(* Logix 5000 project; controller Transcat_L33ER vendor 1 type 14 code 107 rev 32.11; software revision 32.02; part 3 of 5 *)
(* tags used below, declared in another part *)
   AcsiiToReal1 : HexASCII_to_REAL;
   ActiveRecipe : Recipe;   // Active process recipe downloaded from the HMI recipe system and used by the PLC for automatic operation.
   AllDevice1stScanDone : BOOL;   // When this bit is set - all devices have been scanned once and bits reset
   AllDeviceEnable : BOOL;   // A bit to enable or disable the running of all devices
   AllReset : BOOL;   // Bit to reset Auto/Man, AutoRun, RecipeRun, TimedRunEnable to 0 from PLC
   alwaysOFF : BOOL;
   AnyAutoRun : BOOL;   // Bit that in on if ANY device is placed into Auto run (to signal pre-start beed)
   AnyAutoRunFlag : BOOL;   // A flag that indicates if any device is in Auto Run (used with pre-start beep logic)
   AnyManRunFlag : BOOL;   // A flag that indicates if any device is in Manual Run (used with pre-start beep logic)
   AnyManualRun : BOOL;   // Bit that in on if ANY device is placed into manual run (to signal pre-start beed)
   Auto_Run_All_Interlock : BOOL;   // Bit to interlock all devices running in Auto
   AutoRunRequest : BOOL;   // True when the automatic state machine is in RUNNING and automatic device operation is requested.
   Beep : BOOL;   // Bit to Activte Beacon Alarm
   bronkhorstReal : REAL[50];   // data from Bonkhorst - convertred to real values
   BronkOutArr : DINT[3];   // 3 Outputs from Flow controllers 0 - 100% = 0 - 32000
   BronkRealInArr : REAL[100];
   ConversionError : BOOL;
   ConvertedFloat : REAL;
   dataIndex : DINT;   // Bronkhorst Data Index
   Device : Device[20];
   DiscreteTemp : BOOL;   // A temporay boolean to hold positions during PLC transer
   dNum : DINT;   // The index of the current device being processed
   DoseCounter : COUNTER;   // Counts the # of doses since last reset
   DoseCounterReset_HMI : BOOL;   // HMI bit to reset the dose counter
   DoseStart : BOOL;   // Bit to start dosing sequence
   DoseStartOneShot : BOOL;   // One shot to start dosing
   DoseStop : BOOL;   // Bit to stop dosing
   DoseStopOneShot : BOOL;   // one shot to stop dosing
   DoseTarget : REAL;   // Target dose amount
   EstopActive : BOOL;   // E
   EstopFalutResetTOF : TIMER;   // Timer to hold reset bit to allow all drives to reset
   EStopResetPulse : BOOL;   // One-scan pulse used to clear all 14 E-stop interlocks - allows reset of estop interlocks from physical reset button on V
   EStopResetRequired : BOOL;   // Indicates that an estop was actived and it's awaiting reset
   FT103 : BronkhorstFlowMeter;
   FT104 : BronkhorstFlowMeter;
   FT105 : BronkhorstFlowMeter;
   GF101 : Thayer_WB_Feeder;   // Thayer 1 Tags
   GF101_Write_Acknowledge : ALIAS FOR Thayer1_BS:O.Data[2].5;   // Thayer 1 (GF101) Acknowledge
   GF201 : Thayer_WB_Feeder;   // Thayer 2 Tags
   GF201_Totalizer1 : ALIAS FOR Thayer2Data[9];   // Thayer 2 (GF201) Totalizer 1 in lbs
   GF201_Write_Total1Reset : ALIAS FOR Thayer2_BS:O.Data[2].1;   // Thayer 2 (GF1201) Totalizer 1 reset
   HMI_AllReset : BOOL;   // Bit to reset Auto/Man, AutoRun, RecipeRun, TimedRunEnable to 0 from HMI
   HMI_AutoStart : BOOL;   // Starts all devices in AUTO
   HMI_AutoStop : BOOL;   // Stops all devices in AUTO
   HMI_RecipeStart : BOOL;   // Bit to start and stop recipe from HMI
   InitCount : INT;   // Counter to cycle through each device on start-up and reset AutoMan, AutoRun, ManualRun bits
   MX101 : Howes_Mixer;
   MX201 : Howes_Mixer;
   NewDataToggle : BOOL;
   RecipeStart : BOOL;   // Bit to start and stop a recipe execution from PLC logic
   resultIndex : DINT;   // Bronkhorst Real Result Index
   StartBeepTimer : TIMER;   // Timer to sound the beep alarm before starting a device
   TempHexIn : SINT[8];   // Place to copy 8 SINT for proessing by AOI
   TestBit1 : BOOL;   // Just a test bit - does not do anything
   Thayer2ResetTotal1_HMI : BOOL;   // Bit to reset Thayer2 - totalizer 1 from HMI
   VFD_Panel_Safety_Panel_Etop_OK : ALIAS FOR XS26_VFD_Cabinet_Safety_Controller:I1.Data[1].6;
   VFD_Panel_Safety_Remote_Estops_OK : ALIAS FOR XS26_VFD_Cabinet_Safety_Controller:I1.Data[1].7;
(* MainProgram, continued *)

ROUTINE BronkDataMapping   (* structured text *)
// Map FT UDT elements to data to/from Bronkhorst Anybus Gateway
   FT103.AlarmID := Anybus_ETH_SER:I.Data[200];
   FT104.AlarmID := Anybus_ETH_SER:I.Data[201];
   FT105.AlarmID := Anybus_ETH_SER:I.Data[202];
   
   FT103.PV_R := BronkRealInArr[0];
   FT103.TempC := BronkRealInArr[1];
   FT103.Density := BronkRealInArr[2];
   FT103.SP_R := BronkRealInArr[3];
   FT103.Totalizer := BronkRealInArr[4];
   
   FT104.PV_R := BronkRealInArr[5];
   FT104.TempC := BronkRealInArr[6];
   FT104.Density := BronkRealInArr[7];
   FT104.SP_R := BronkRealInArr[8];
   FT104.Totalizer := BronkRealInArr[9];
   
   FT105.PV_R := BronkRealInArr[10];
   FT105.TempC := BronkRealInArr[11];
   FT105.Density := BronkRealInArr[12];
   FT105.SP_R := BronkRealInArr[13];
   FT105.Totalizer := BronkRealInArr[14];
   
   FT103.OT_R := (BronkOutArr[0]) / 167681.5;
   FT104.OT_R := (BronkOutArr[1]) / 167681.5;
   FT105.OT_R := (BronkOutArr[2]) / 167681.5;
END_ROUTINE

ROUTINE Bronkhorst_Data   (* ladder *)
// read and write data to/from the EIP instance and convert to/from 8 byte to/from floating point
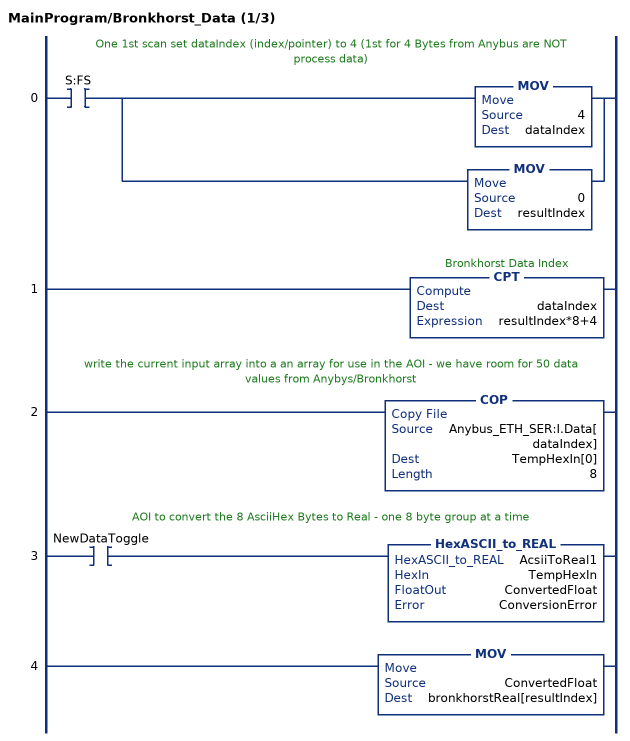
   // One 1st scan set dataIndex (index/pointer) to 4 (1st for 4 Bytes from Anybus are NOT process data)
   0: XIC(S:FS)[MOV(4,dataIndex) ,MOV(0,resultIndex) ];
   1: CPT(dataIndex,resultIndex*8+4);
   // write the current input array into a an array for use in the AOI - we have room for 50 data values from Anybys/Bronkhorst
   2: COP(Anybus_ETH_SER:I.Data[dataIndex],TempHexIn[0],8);
   // AOI to convert the 8 AsciiHex Bytes to Real - one 8 byte group at a time
   3: XIC(NewDataToggle)HexASCII_to_REAL(AcsiiToReal1,TempHexIn,ConvertedFloat,ConversionError);
   4: MOV(ConvertedFloat,bronkhorstReal[resultIndex]);
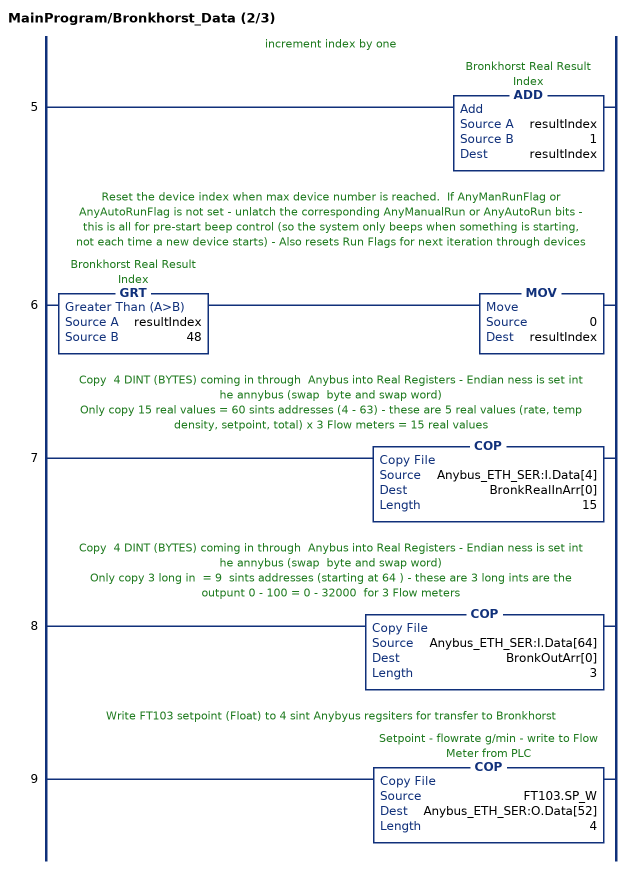
   // increment index by one
   5: ADD(resultIndex,1,resultIndex);
   // Reset the device index when max device number is reached.  If AnyManRunFlag or AnyAutoRunFlag is not set - unlatch the corresponding AnyManualRun or AnyAutoRun bits - this is all for pre-start beep control (so the system only beeps when something is starting, not each time a new device starts) - Also resets Run Flags for next iteration through devices
   6: GRT(resultIndex,48)MOV(0,resultIndex);
   // Copy  4 DINT (BYTES) coming in through  Anybus into Real Registers - Endian ness is set int he annybus (swap  byte and swap word)
   // Only copy 15 real values = 60 sints addresses (4 - 63) - these are 5 real values (rate, temp density, setpoint, total) x 3 Flow meters = 15 real values
   7: COP(Anybus_ETH_SER:I.Data[4],BronkRealInArr[0],15);
   // Copy  4 DINT (BYTES) coming in through  Anybus into Real Registers - Endian ness is set int he annybus (swap  byte and swap word)
   // Only copy 3 long in  = 9  sints addresses (starting at 64 ) - these are 3 long ints are the outpunt 0 - 100 = 0 - 32000  for 3 Flow meters
   8: COP(Anybus_ETH_SER:I.Data[64],BronkOutArr[0],3);
   // Write FT103 setpoint (Float) to 4 sint Anybyus regsiters for transfer to Bronkhorst
   9: COP(FT103.SP_W,Anybus_ETH_SER:O.Data[52],4);
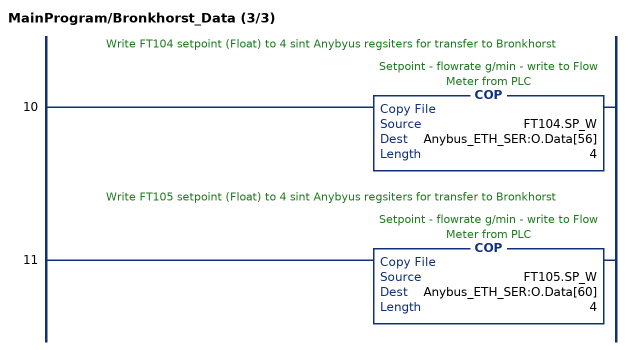
   // Write FT104 setpoint (Float) to 4 sint Anybyus regsiters for transfer to Bronkhorst
   10: COP(FT104.SP_W,Anybus_ETH_SER:O.Data[56],4);
   // Write FT105 setpoint (Float) to 4 sint Anybyus regsiters for transfer to Bronkhorst
   11: COP(FT105.SP_W,Anybus_ETH_SER:O.Data[60],4);
END_ROUTINE

ROUTINE DeviceLogic   (* ladder *)
// Process the logic for each device with index and indirect addressing.
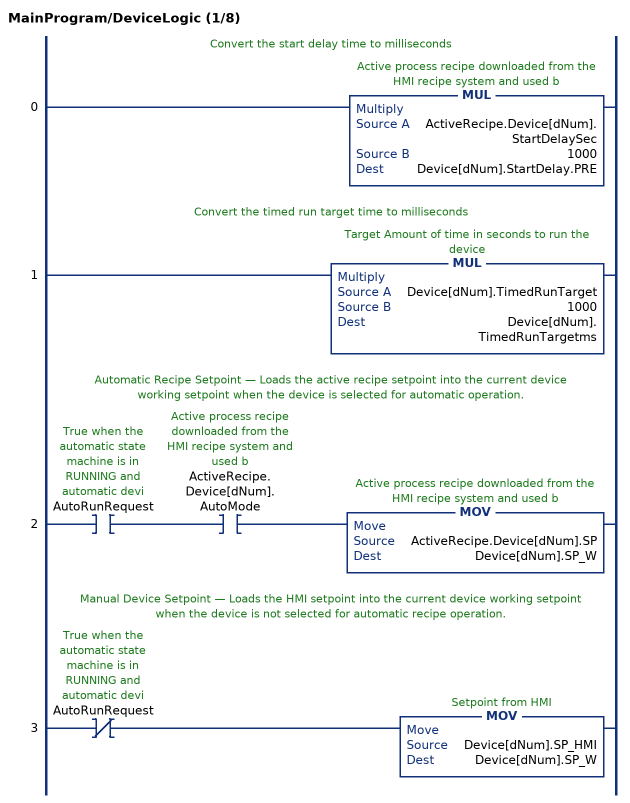
   // Convert the start delay time to milliseconds
   0: MUL(ActiveRecipe.Device[dNum].StartDelaySec,1000,Device[dNum].StartDelay.PRE);
   // Convert the timed run target time to milliseconds
   1: MUL(Device[dNum].TimedRunTarget,1000,Device[dNum].TimedRunTargetms);
   // Automatic Recipe Setpoint — Loads the active recipe setpoint into the current device working setpoint when the device is selected for automatic operation.
   2: XIC(AutoRunRequest)XIC(ActiveRecipe.Device[dNum].AutoMode)MOV(ActiveRecipe.Device[dNum].SP,Device[dNum].SP_W);
   // Manual Device Setpoint — Loads the HMI setpoint into the current device working setpoint when the device is not selected for automatic recipe operation.
   3: XIO(AutoRunRequest)MOV(Device[dNum].SP_HMI,Device[dNum].SP_W);
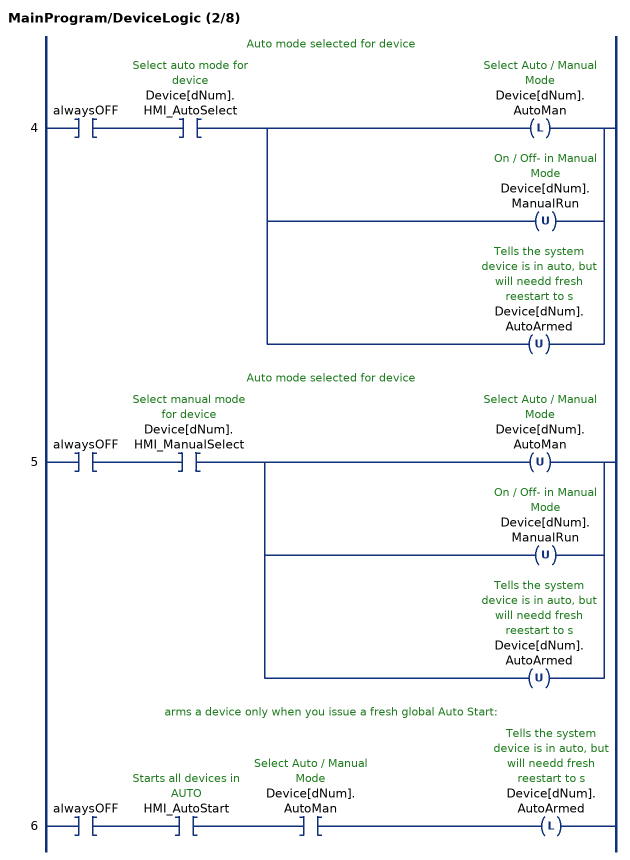
   // Auto mode selected for device
   4: XIC(alwaysOFF)XIC(Device[dNum].HMI_AutoSelect)[OTL(Device[dNum].AutoMan) ,OTU(Device[dNum].ManualRun) ,OTU(Device[dNum].AutoArmed) ];
   // Auto mode selected for device
   5: XIC(alwaysOFF)XIC(Device[dNum].HMI_ManualSelect)[OTU(Device[dNum].AutoMan) ,[OTU(Device[dNum].ManualRun) ,OTU(Device[dNum].AutoArmed) ] ];
   // arms a device only when you issue a fresh global Auto Start:
   6: XIC(alwaysOFF)XIC(HMI_AutoStart)XIC(Device[dNum].AutoMan)OTL(Device[dNum].AutoArmed);
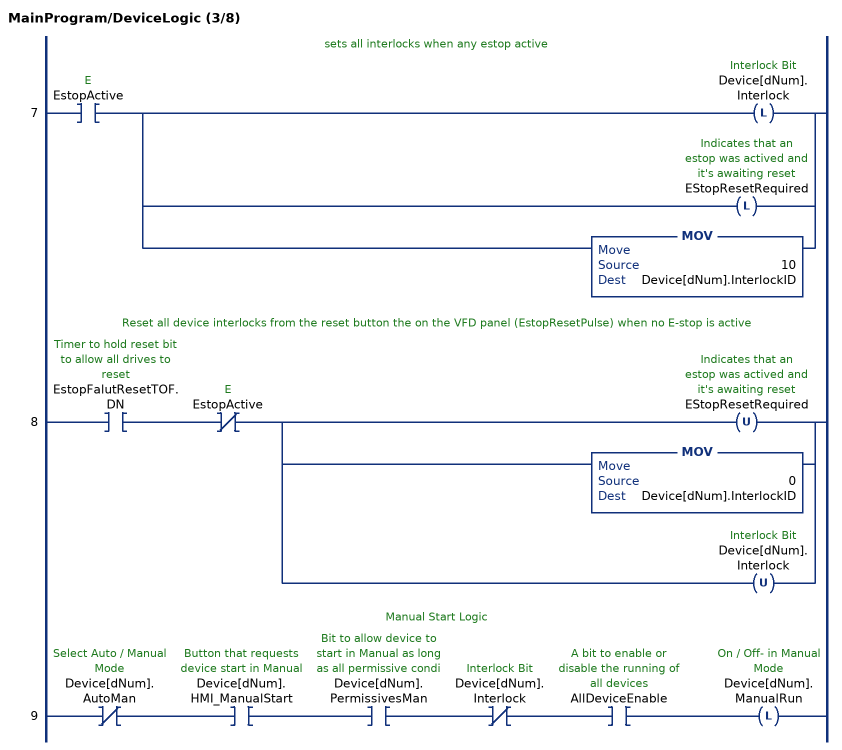
   // sets all interlocks when any estop active
   7: XIC(EstopActive)[OTL(Device[dNum].Interlock) ,OTL(EStopResetRequired) ,MOV(10,Device[dNum].InterlockID) ];
   // Reset all device interlocks from the reset button the on the VFD panel (EstopResetPulse) when no E-stop is active
   8: XIC(EstopFalutResetTOF.DN)XIO(EstopActive)[OTU(EStopResetRequired) ,MOV(0,Device[dNum].InterlockID) ,OTU(Device[dNum].Interlock) ];
   // Manual Start Logic
   9: XIO(Device[dNum].AutoMan)XIC(Device[dNum].HMI_ManualStart)XIC(Device[dNum].PermissivesMan)XIO(Device[dNum].Interlock)XIC(AllDeviceEnable)OTL(Device[dNum].ManualRun);
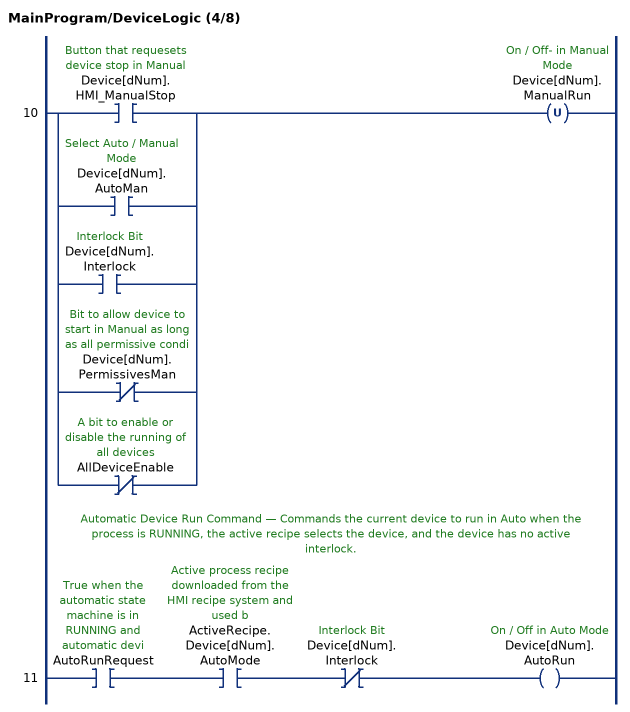
   10: [XIC(Device[dNum].HMI_ManualStop) ,[XIC(Device[dNum].AutoMan) ,[XIC(Device[dNum].Interlock) ,[XIO(Device[dNum].PermissivesMan) ,XIO(AllDeviceEnable) ] ] ] ]OTU(Device[dNum].ManualRun);
   // Automatic Device Run Command — Commands the current device to run in Auto when the process is RUNNING, the active recipe selects the device, and the device has no active interlock.
   11: XIC(AutoRunRequest)XIC(ActiveRecipe.Device[dNum].AutoMode)XIO(Device[dNum].Interlock)OTE(Device[dNum].AutoRun);
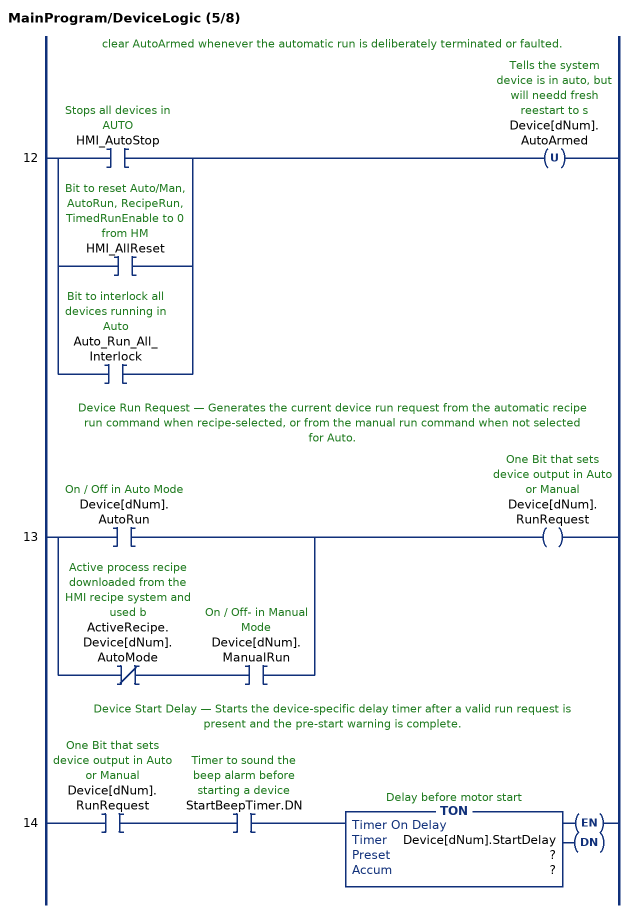
   // clear AutoArmed whenever the automatic run is deliberately terminated or faulted.
   12: [XIC(HMI_AutoStop) ,[XIC(HMI_AllReset) ,XIC(Auto_Run_All_Interlock) ] ]OTU(Device[dNum].AutoArmed);
   // Device Run Request — Generates the current device run request from the automatic recipe run command when recipe-selected, or from the manual run command when not selected for Auto.
   13: [XIC(Device[dNum].AutoRun) ,XIO(ActiveRecipe.Device[dNum].AutoMode) XIC(Device[dNum].ManualRun) ]OTE(Device[dNum].RunRequest);
   // Device Start Delay — Starts the device-specific delay timer after a valid run request is present and the pre-start warning is complete.
   14: XIC(Device[dNum].RunRequest)XIC(StartBeepTimer.DN)TON(Device[dNum].StartDelay,?,?);
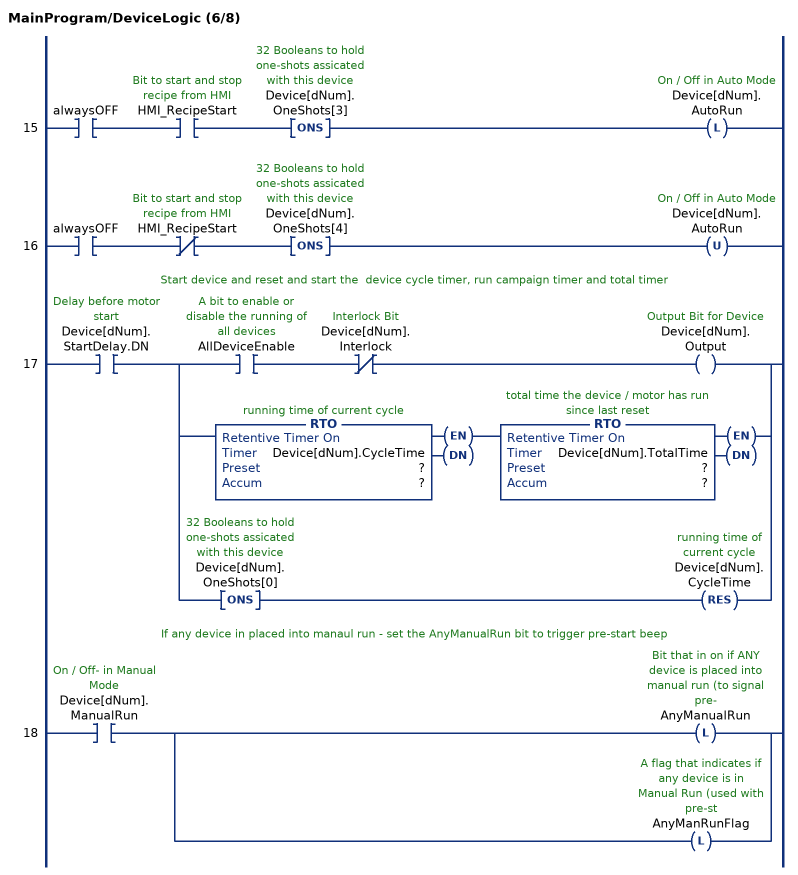
   15: XIC(alwaysOFF)XIC(HMI_RecipeStart)ONS(Device[dNum].OneShots[3])OTL(Device[dNum].AutoRun);
   16: XIC(alwaysOFF)XIO(HMI_RecipeStart)ONS(Device[dNum].OneShots[4])OTU(Device[dNum].AutoRun);
   // Start device and reset and start the  device cycle timer, run campaign timer and total timer
   17: XIC(Device[dNum].StartDelay.DN)[XIC(AllDeviceEnable) XIO(Device[dNum].Interlock) OTE(Device[dNum].Output) ,[RTO(Device[dNum].CycleTime,?,?) RTO(Device[dNum].TotalTime,?,?) ,ONS(Device[dNum].OneShots[0]) RES(Device[dNum].CycleTime) ] ];
   // If any device in placed into manaul run - set the AnyManualRun bit to trigger pre-start beep
   18: XIC(Device[dNum].ManualRun)[OTL(AnyManualRun) ,OTL(AnyManRunFlag) ];
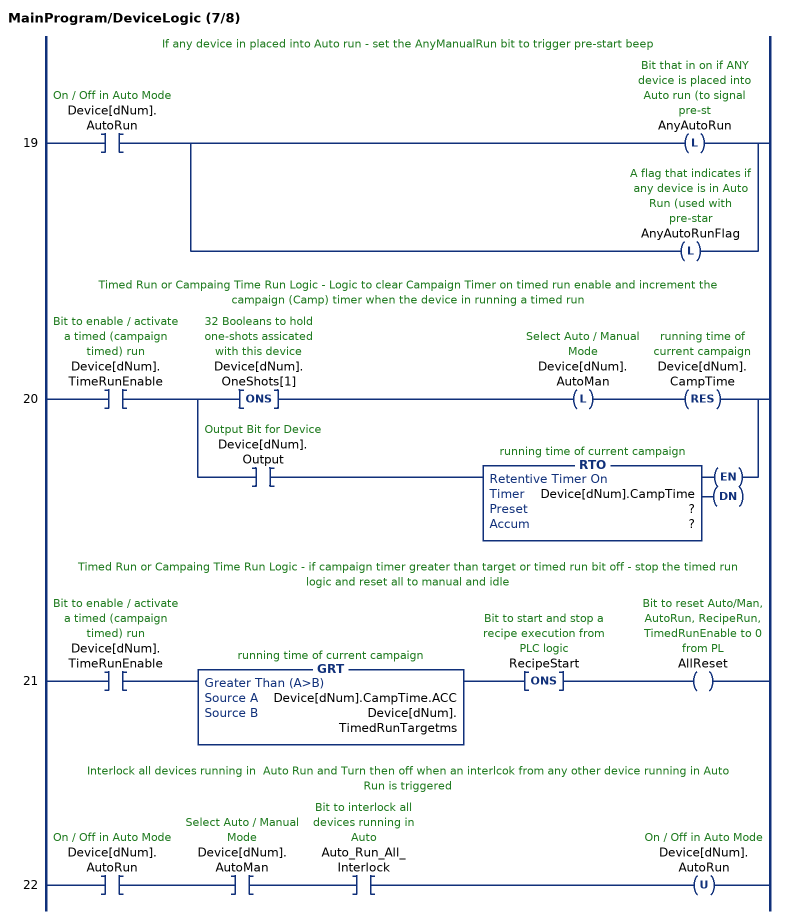
   // If any device in placed into Auto run - set the AnyManualRun bit to trigger pre-start beep
   19: XIC(Device[dNum].AutoRun)[OTL(AnyAutoRun) ,OTL(AnyAutoRunFlag) ];
   // Timed Run or Campaing Time Run Logic - Logic to clear Campaign Timer on timed run enable and increment the campaign (Camp) timer when the device in running a timed run
   20: XIC(Device[dNum].TimeRunEnable)[ONS(Device[dNum].OneShots[1]) OTL(Device[dNum].AutoMan) RES(Device[dNum].CampTime) ,XIC(Device[dNum].Output) RTO(Device[dNum].CampTime,?,?) ];
   // Timed Run or Campaing Time Run Logic - if campaign timer greater than target or timed run bit off - stop the timed run logic and reset all to manual and idle
   21: XIC(Device[dNum].TimeRunEnable)GRT(Device[dNum].CampTime.ACC,Device[dNum].TimedRunTargetms)ONS(RecipeStart)OTE(AllReset);
   // Interlock all devices running in  Auto Run and Turn then off when an interlcok from any other device running in Auto Run is triggered
   22: XIC(Device[dNum].AutoRun)XIC(Device[dNum].AutoMan)XIC(Auto_Run_All_Interlock)OTU(Device[dNum].AutoRun);
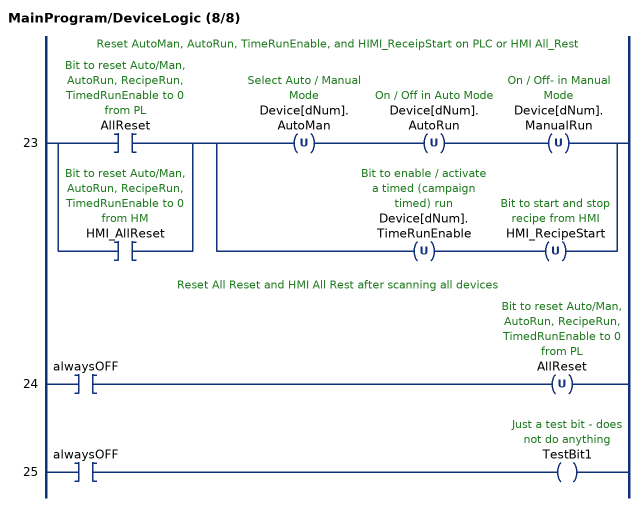
   // Reset AutoMan, AutoRun, TimeRunEnable, and HIMI_ReceipStart on PLC or HMI All_Rest
   23: [XIC(AllReset) ,XIC(HMI_AllReset) ][OTU(Device[dNum].AutoMan) OTU(Device[dNum].AutoRun) OTU(Device[dNum].ManualRun) ,OTU(Device[dNum].TimeRunEnable) OTU(HMI_RecipeStart) ];
   // Reset All Reset and HMI All Rest after scanning all devices
   24: XIC(alwaysOFF)OTU(AllReset);
   25: XIC(alwaysOFF)OTE(TestBit1);
END_ROUTINE

ROUTINE DeviceManager   (* ladder *)
// Loop through all devices each scan
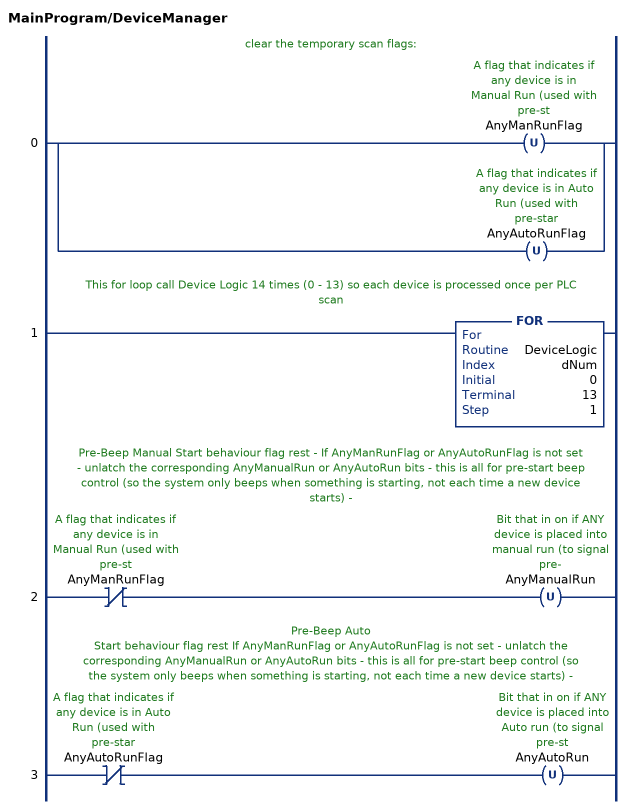
   // clear the temporary scan flags:
   0: [OTU(AnyManRunFlag) ,OTU(AnyAutoRunFlag) ];
   // This for loop call Device Logic 14 times (0 - 13) so each device is processed once per PLC scan
   1: FOR(DeviceLogic,dNum,0,13,1);
   // Pre-Beep Manual Start behaviour flag rest - If AnyManRunFlag or AnyAutoRunFlag is not set - unlatch the corresponding AnyManualRun or AnyAutoRun bits - this is all for pre-start beep control (so the system only beeps when something is starting, not each time a new device starts) -
   2: XIO(AnyManRunFlag)OTU(AnyManualRun);
   // Pre-Beep Auto
   //  Start behaviour flag rest If AnyManRunFlag or AnyAutoRunFlag is not set - unlatch the corresponding AnyManualRun or AnyAutoRun bits - this is all for pre-start beep control (so the system only beeps when something is starting, not each time a new device starts) -
   3: XIO(AnyAutoRunFlag)OTU(AnyAutoRun);
END_ROUTINE

ROUTINE GF201Dose   (* ladder *)
// Logic to Dose a specific amount from GF201 - Thayer 2
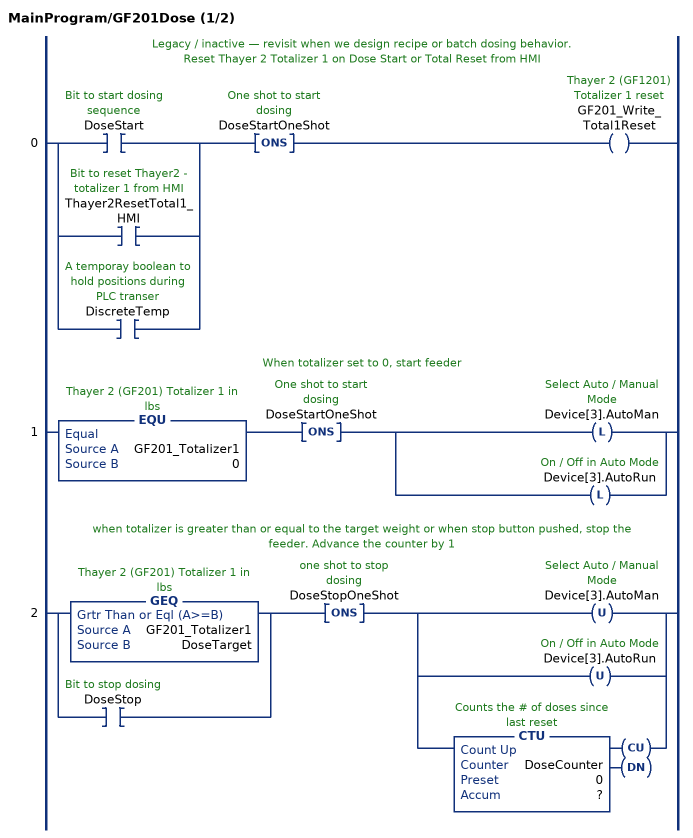
   // Legacy / inactive — revisit when we design recipe or batch dosing behavior.
   // Reset Thayer 2 Totalizer 1 on Dose Start or Total Reset from HMI
   0: [XIC(DoseStart) ,[XIC(Thayer2ResetTotal1_HMI) ,XIC(DiscreteTemp) ] ]ONS(DoseStartOneShot)OTE(GF201_Write_Total1Reset);
   // When totalizer set to 0, start feeder
   1: EQU(GF201_Totalizer1,0)ONS(DoseStartOneShot)[OTL(Device[3].AutoMan) ,OTL(Device[3].AutoRun) ];
   // when totalizer is greater than or equal to the target weight or when stop button pushed, stop the feeder. Advance the counter by 1
   2: [GEQ(GF201_Totalizer1,DoseTarget) ,XIC(DoseStop) ]ONS(DoseStopOneShot)[OTU(Device[3].AutoMan) ,[OTU(Device[3].AutoRun) ,CTU(DoseCounter,?,?) ] ];
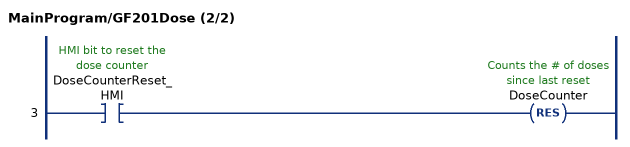
   3: XIC(DoseCounterReset_HMI)RES(DoseCounter);
END_ROUTINE

ROUTINE Initialize   (* ladder *)
// Reset controls and any other initialization required
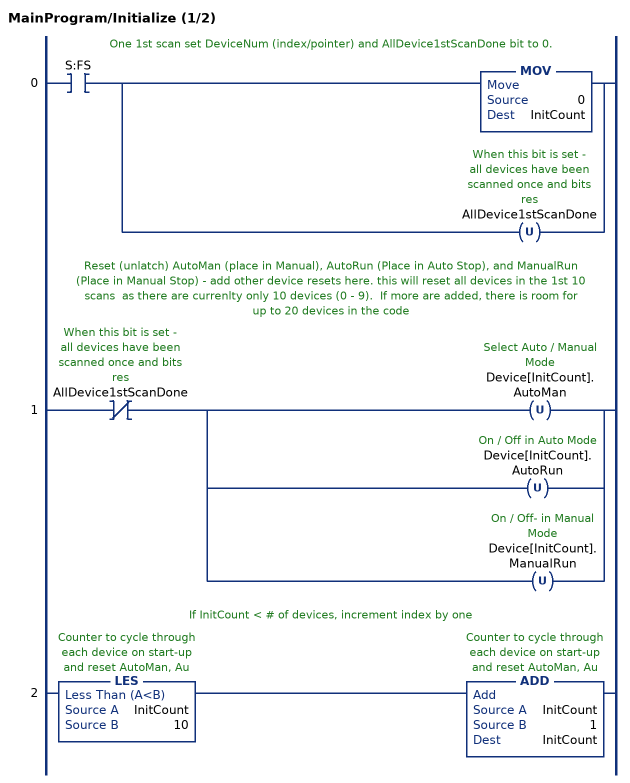
   // One 1st scan set DeviceNum (index/pointer) and AllDevice1stScanDone bit to 0.
   0: XIC(S:FS)[MOV(0,InitCount) ,OTU(AllDevice1stScanDone) ];
   // Reset (unlatch) AutoMan (place in Manual), AutoRun (Place in Auto Stop), and ManualRun (Place in Manual Stop) - add other device resets here. this will reset all devices in the 1st 10 scans  as there are currenlty only 10 devices (0 - 9).  If more are added, there is room for up to 20 devices in the code
   1: XIO(AllDevice1stScanDone)[OTU(Device[InitCount].AutoMan) ,[OTU(Device[InitCount].AutoRun) ,OTU(Device[InitCount].ManualRun) ] ];
   // If InitCount < # of devices, increment index by one
   2: LES(InitCount,10)ADD(InitCount,1,InitCount);
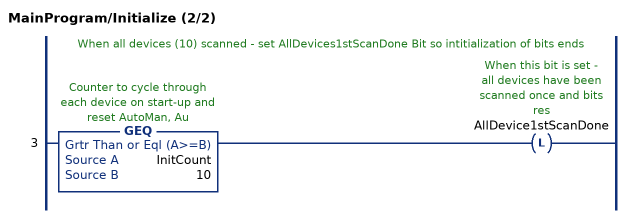
   // When all devices (10) scanned - set AllDevices1stScanDone Bit so intitialization of bits ends
   3: GEQ(InitCount,10)OTL(AllDevice1stScanDone);
END_ROUTINE

ROUTINE InterlockLogic   (* ladder *)
// All interlock logic is handled here
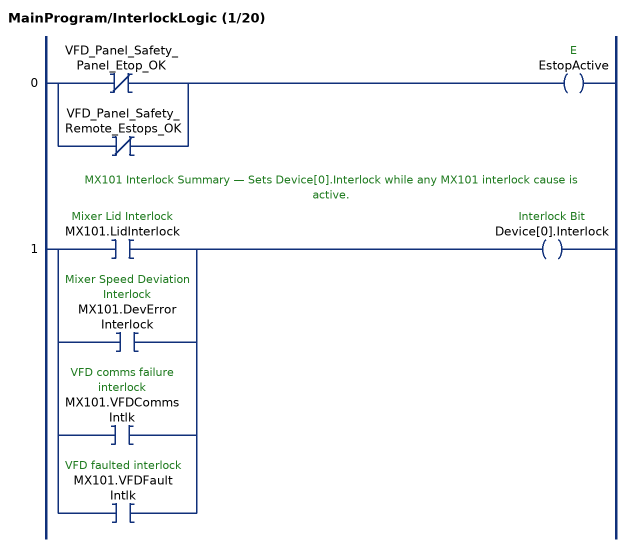
   0: [XIO(VFD_Panel_Safety_Panel_Etop_OK) ,XIO(VFD_Panel_Safety_Remote_Estops_OK) ]OTE(EstopActive);
   // MX101 Interlock Summary — Sets Device[0].Interlock while any MX101 interlock cause is active.
   1: [XIC(MX101.LidInterlock) ,XIC(MX101.DevErrorInterlock) ,XIC(MX101.VFDCommsIntlk) ,XIC(MX101.VFDFaultIntlk) ]OTE(Device[0].Interlock);
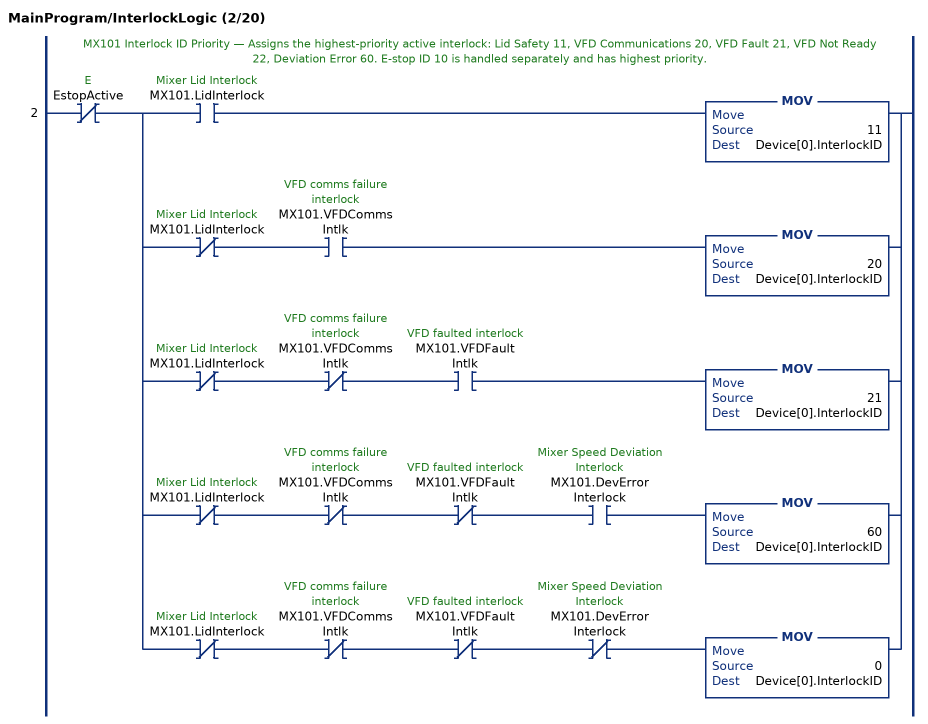
   // MX101 Interlock ID Priority — Assigns the highest-priority active interlock: Lid Safety 11, VFD Communications 20, VFD Fault 21, VFD Not Ready 22, Deviation Error 60. E-stop ID 10 is handled separately and has highest priority.
   2: XIO(EstopActive)[XIC(MX101.LidInterlock) MOV(11,Device[0].InterlockID) ,XIO(MX101.LidInterlock) XIC(MX101.VFDCommsIntlk) MOV(20,Device[0].InterlockID) ,XIO(MX101.LidInterlock) XIO(MX101.VFDCommsIntlk) XIC(MX101.VFDFaultIntlk) MOV(21,Device[0].InterlockID) ,XIO(MX101.LidInterlock) XIO(MX101.VFDCommsIntlk) XIO(MX101.VFDFaultIntlk) XIC(MX101.DevErrorInterlock) MOV(60,Device[0].InterlockID) ,XIO(MX101.LidInterlock) XIO(MX101.VFDCommsIntlk) XIO(MX101.VFDFaultIntlk) XIO(MX101.DevErrorInterlock) MOV(0,Device[0].InterlockID) ];
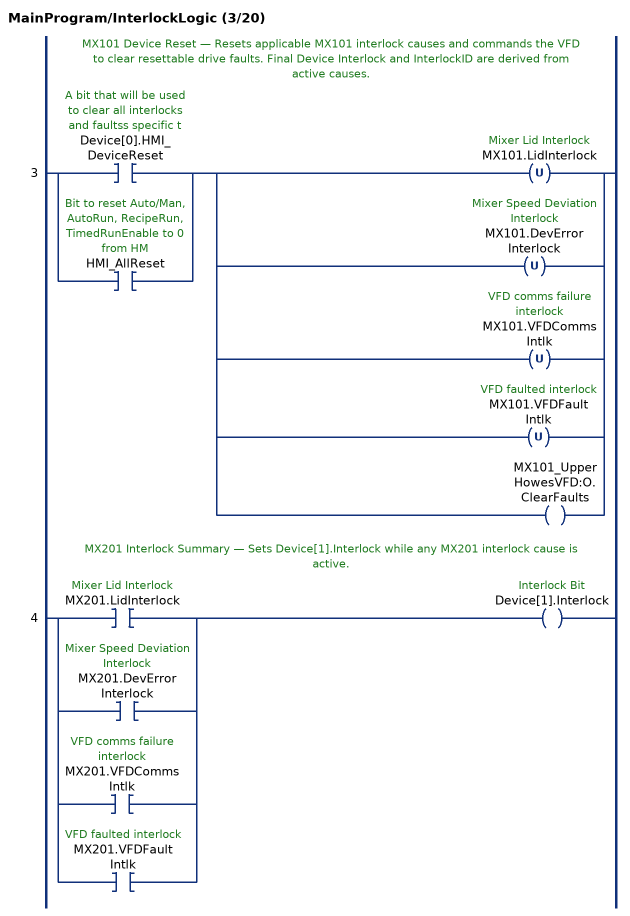
   // MX101 Device Reset — Resets applicable MX101 interlock causes and commands the VFD to clear resettable drive faults. Final Device Interlock and InterlockID are derived from active causes.
   3: [XIC(Device[0].HMI_DeviceReset) ,XIC(HMI_AllReset) ][OTU(MX101.LidInterlock) ,OTU(MX101.DevErrorInterlock) ,OTU(MX101.VFDCommsIntlk) ,OTU(MX101.VFDFaultIntlk) ,OTE(MX101_UpperHowesVFD:O.ClearFaults) ];
   // MX201 Interlock Summary — Sets Device[1].Interlock while any MX201 interlock cause is active.
   4: [XIC(MX201.LidInterlock) ,XIC(MX201.DevErrorInterlock) ,XIC(MX201.VFDCommsIntlk) ,XIC(MX201.VFDFaultIntlk) ]OTE(Device[1].Interlock);
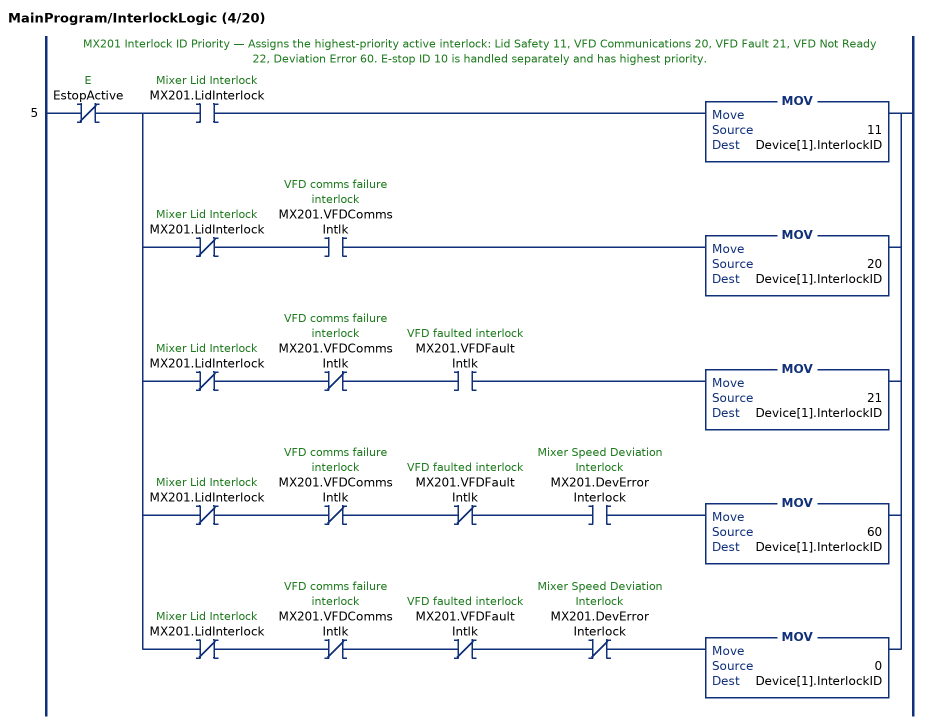
   // MX201 Interlock ID Priority — Assigns the highest-priority active interlock: Lid Safety 11, VFD Communications 20, VFD Fault 21, VFD Not Ready 22, Deviation Error 60. E-stop ID 10 is handled separately and has highest priority.
   5: XIO(EstopActive)[XIC(MX201.LidInterlock) MOV(11,Device[1].InterlockID) ,XIO(MX201.LidInterlock) XIC(MX201.VFDCommsIntlk) MOV(20,Device[1].InterlockID) ,XIO(MX201.LidInterlock) XIO(MX201.VFDCommsIntlk) XIC(MX201.VFDFaultIntlk) MOV(21,Device[1].InterlockID) ,XIO(MX201.LidInterlock) XIO(MX201.VFDCommsIntlk) XIO(MX201.VFDFaultIntlk) XIC(MX201.DevErrorInterlock) MOV(60,Device[1].InterlockID) ,XIO(MX201.LidInterlock) XIO(MX201.VFDCommsIntlk) XIO(MX201.VFDFaultIntlk) XIO(MX201.DevErrorInterlock) MOV(0,Device[1].InterlockID) ];
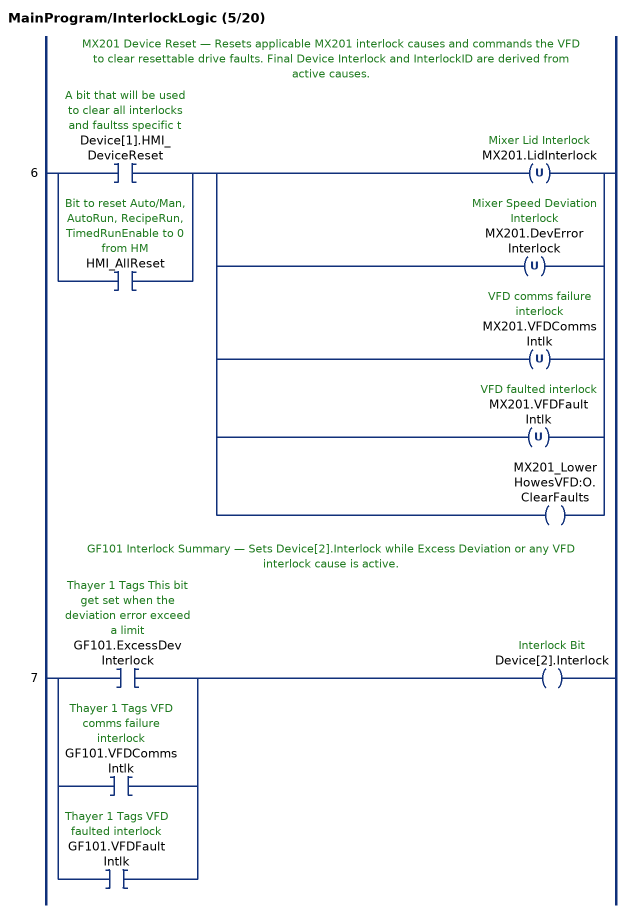
   // MX201 Device Reset — Resets applicable MX201 interlock causes and commands the VFD to clear resettable drive faults. Final Device Interlock and InterlockID are derived from active causes.
   6: [XIC(Device[1].HMI_DeviceReset) ,XIC(HMI_AllReset) ][OTU(MX201.LidInterlock) ,OTU(MX201.DevErrorInterlock) ,OTU(MX201.VFDCommsIntlk) ,OTU(MX201.VFDFaultIntlk) ,OTE(MX201_LowerHowesVFD:O.ClearFaults) ];
   // GF101 Interlock Summary — Sets Device[2].Interlock while Excess Deviation or any VFD interlock cause is active.
   7: [XIC(GF101.ExcessDevInterlock) ,XIC(GF101.VFDCommsIntlk) ,XIC(GF101.VFDFaultIntlk) ]OTE(Device[2].Interlock);
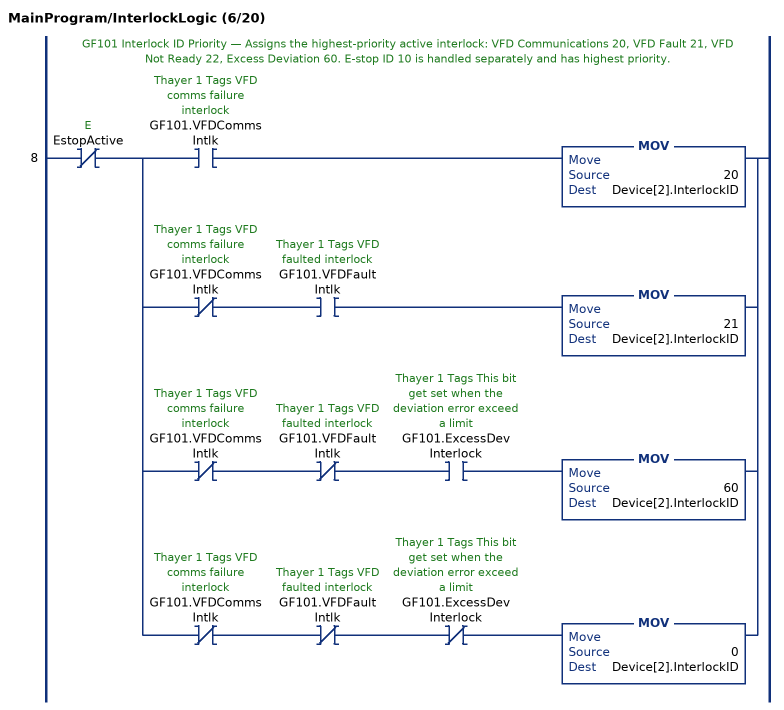
   // GF101 Interlock ID Priority — Assigns the highest-priority active interlock: VFD Communications 20, VFD Fault 21, VFD Not Ready 22, Excess Deviation 60. E-stop ID 10 is handled separately and has highest priority.
   8: XIO(EstopActive)[XIC(GF101.VFDCommsIntlk) MOV(20,Device[2].InterlockID) ,XIO(GF101.VFDCommsIntlk) XIC(GF101.VFDFaultIntlk) MOV(21,Device[2].InterlockID) ,XIO(GF101.VFDCommsIntlk) XIO(GF101.VFDFaultIntlk) XIC(GF101.ExcessDevInterlock) MOV(60,Device[2].InterlockID) ,XIO(GF101.VFDCommsIntlk) XIO(GF101.VFDFaultIntlk) XIO(GF101.ExcessDevInterlock) MOV(0,Device[2].InterlockID) ];
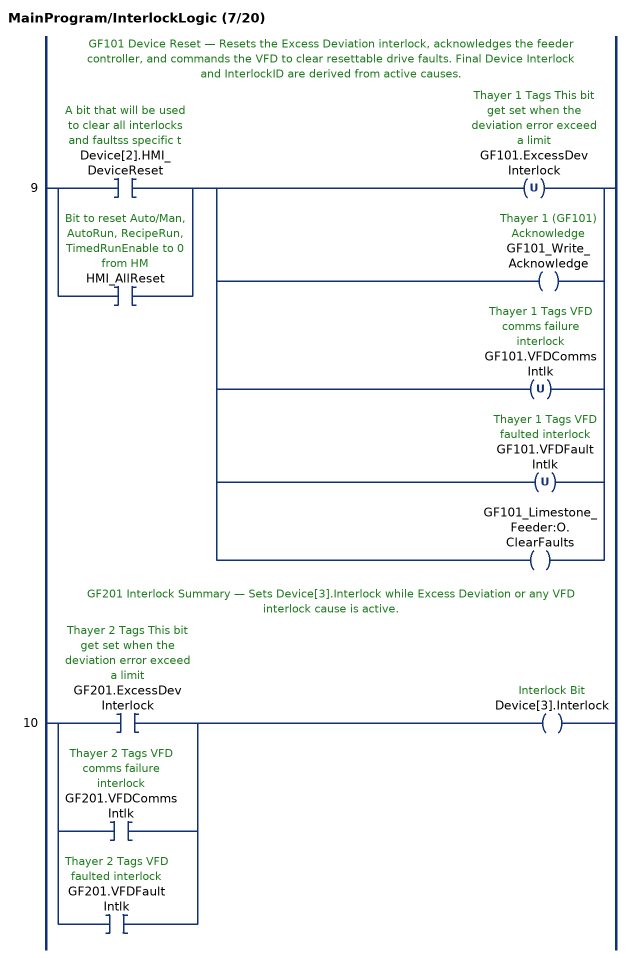
   // GF101 Device Reset — Resets the Excess Deviation interlock, acknowledges the feeder controller, and commands the VFD to clear resettable drive faults. Final Device Interlock and InterlockID are derived from active causes.
   9: [XIC(Device[2].HMI_DeviceReset) ,XIC(HMI_AllReset) ][OTU(GF101.ExcessDevInterlock) ,OTE(GF101_Write_Acknowledge) ,OTU(GF101.VFDCommsIntlk) ,OTU(GF101.VFDFaultIntlk) ,OTE(GF101_Limestone_Feeder:O.ClearFaults) ];
   // GF201 Interlock Summary — Sets Device[3].Interlock while Excess Deviation or any VFD interlock cause is active.
   10: [XIC(GF201.ExcessDevInterlock) ,XIC(GF201.VFDCommsIntlk) ,XIC(GF201.VFDFaultIntlk) ]OTE(Device[3].Interlock);
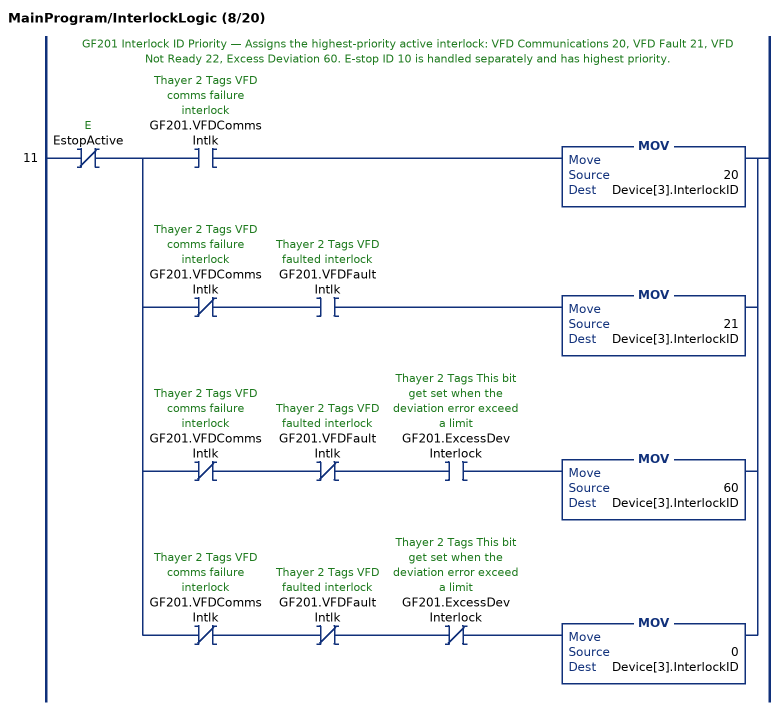
   // GF201 Interlock ID Priority — Assigns the highest-priority active interlock: VFD Communications 20, VFD Fault 21, VFD Not Ready 22, Excess Deviation 60. E-stop ID 10 is handled separately and has highest priority.
   11: XIO(EstopActive)[XIC(GF201.VFDCommsIntlk) MOV(20,Device[3].InterlockID) ,XIO(GF201.VFDCommsIntlk) XIC(GF201.VFDFaultIntlk) MOV(21,Device[3].InterlockID) ,XIO(GF201.VFDCommsIntlk) XIO(GF201.VFDFaultIntlk) XIC(GF201.ExcessDevInterlock) MOV(60,Device[3].InterlockID) ,XIO(GF201.VFDCommsIntlk) XIO(GF201.VFDFaultIntlk) XIO(GF201.ExcessDevInterlock) MOV(0,Device[3].InterlockID) ];
